FUNCTION_BLOCK MachineSequence EXTENDS ZApplication.Sequence
VAR
  {attribute 'hide'}
  _parent : REFERENCE TO MachineUnit;
  _io : REFERENCE TO MachineIo;
  _actuator : REFERENCE TO MachineActuator;
  _fieldbus : REFERENCE TO MachineFieldbus;
  _axis : REFERENCE TO MachineAxis;
  _data : REFERENCE TO MachineDataRef;
  _unit : REFERENCE TO MachineLinkedUnit;  
END_VAR

METHOD FB_init : BOOL
VAR_INPUT
  bInitRetains : BOOL; // if TRUE, the retain variables are initialized (warm start / cold start)
  bInCopyCode : BOOL;  // if TRUE, the instance afterwards gets moved into the copy code (online change)
  unit : REFERENCE TO MachineUnit;
END_VAR
_parent REF= unit;
_alarming := unit._alarming;
_io REF= unit._equipment.Io;
_actuator REF= unit._equipment.Actuator;
_fieldbus REF= unit._equipment.Fieldbus;
_axis REF= unit._equipment.Axis;
_unit REF= unit._equipment.Unit;
_data REF= unit._data;
_loggerDiagnostics.SetLogger(unit._logger);
END_METHOD

METHOD StepDecoded : ZCore.ZString
VAR_INPUT
  stepIndex : INT;
END_VAR
VAR_INST
  _stepIndexDecoded : MachineStep;
END_VAR
_stepIndexDecoded := stepIndex;
stepDecoded := TO_STRING(_stepIndexDecoded);
END_METHOD

END_FUNCTION_BLOCK

(* stored: Version 1.1.0.1
   POU MachineSequence: Id {4d32c1fd-5c0e-4032-a876-8c1b86464b27}, SpecialFunc None
   Method FB_init: Id {29884392-ac60-459d-8bce-1747dd1601bc}
   Method StepDecoded: Id {923180d7-ccf5-48cb-8ede-1a7e1b7bbcd7} *)
